// TIA Portal project "SortingStation" (V17)

(* hardware
DEVICE "S7-1500/ET200MP station_1"  S7-1500 station
   slot 0: "Rail_0"  Rack  6ES7 590-1***0-0AA0
   slot 1: "PLC_1"  CPU 1511-1 PN  6ES7 511-1AK02-0AB0  V2.9
      slot 3: "CPU display_1"  6ES7591-1AA00-0AA0
      slot 32768: "PROFINET interface_1"  X1
         slot 32769: "Port_1"  X1 P1
         slot 32770: "Port_2"  X1 P2
      slot 34817: "Virtual CP interface port_1"  Virtual CP interface port  Virtual CP interface port
   slot 2: "DI 16x24VDC BA_1"  DI 16x24VDC BA  6ES7 521-1BH10-0AA0  V1.1
   slot 3: "DQ 16x24VDC/0.5A BA_1"  DQ 16x24VDC/0.5A BA  6ES7 522-1BH10-0AA0  V1.1
   slot 4: "AI 4xU/I/RTD/TC ST_1"  AI 4xU/I/RTD/TC ST  6ES7 531-7QD00-0AB0  V1.0
   slot 5: "AQ 4xU/I ST_1"  AQ 4xU/I ST  6ES7 532-5HD00-0AB0  V2.2
*)

// ===== PLC "PLC_1"  CPU 1511-1 PN =====

VAR_GLOBAL   // PLC tag table "Default tag table"
   "System_Byte" AT %MB1 : Byte;
   "FirstScan" AT %M1.0 : Bool;
   "DiagStatusUpdate" AT %M1.1 : Bool;
   "AlwaysTRUE" AT %M1.2 : Bool;
   "AlwaysFALSE" AT %M1.3 : Bool;
   "Clock_Byte" AT %MB0 : Byte;
   "Clock_10Hz" AT %M0.0 : Bool;
   "Clock_5Hz" AT %M0.1 : Bool;
   "Clock_2.5Hz" AT %M0.2 : Bool;
   "Clock_2Hz" AT %M0.3 : Bool;
   "Clock_1.25Hz" AT %M0.4 : Bool;
   "Clock_1Hz" AT %M0.5 : Bool;
   "Clock_0.625Hz" AT %M0.6 : Bool;
   "Clock_0.5Hz" AT %M0.7 : Bool;
END_VAR

VAR_GLOBAL   // PLC tag table "io"
   "At exit" AT %I0.0 : Bool;
   "Counter 1" AT %QD30 : DInt;
   "Vision sensor" AT %ID30 : DInt;
   "Remover 3" AT %Q1.7 : Bool;
   "Remover 2" AT %Q1.6 : Bool;
   "Remover 1" AT %Q1.5 : Bool;
   "Emitter" AT %Q1.4 : Bool;
   "Stop light" AT %Q1.3 : Bool;
   "Reset light" AT %Q1.2 : Bool;
   "Start light" AT %Q1.1 : Bool;
   "Sorter 3 belt" AT %Q1.0 : Bool;
   "Sorter 3 turn" AT %Q0.7 : Bool;
   "Sorter 2 belt" AT %Q0.6 : Bool;
   "Sorter 2 turn" AT %Q0.5 : Bool;
   "Sorter 1 belt" AT %Q0.4 : Bool;
   "Sorter 1 turn" AT %Q0.3 : Bool;
   "Exit conveyor" AT %Q0.2 : Bool;
   "Stop blade" AT %Q0.1 : Bool;
   "Entry conveyor" AT %Q0.0 : Bool;
   "Manual" AT %I0.7 : Bool;
   "FACTORY I/O (Running)" AT %I0.6 : Bool;
   "Auto" AT %I0.5 : Bool;
   "Emergency stop" AT %I0.4 : Bool;
   "Stop" AT %I0.3 : Bool;
   "Reset" AT %I0.2 : Bool;
   "Start" AT %I0.1 : Bool;
   "Counter 2" AT %QD34 : DInt;
   "Counter 3" AT %QD38 : DInt;
END_VAR

DATA_BLOCK "HmiData"   // DB1
{ S7_Optimized_Access := 'TRUE' }
VERSION : 0.1
   VAR
      Flank : Bool;
      Flank_1 : Bool;
      Flank_2 : Bool;
      Flank_3 : Bool;
      Flank_4 : Bool;
      reset1 : Bool;
      reset2 : Bool;
      reset3 : Bool;
   END_VAR
BEGIN
END_DATA_BLOCK

// folder: System blocks/Program resources

DATA_BLOCK "IEC_Counter_0_DB_3"   // DB5
{ S7_Optimized_Access := 'TRUE' }
AUTHOR : Simatic
FAMILY : IEC
NAME : CNTR
VERSION : 1.0
// stored: InstanceOfName IEC_COUNTER
"IEC_COUNTER"
BEGIN
END_DATA_BLOCK

DATA_BLOCK "IEC_Counter_0_DB_4"   // DB6
{ S7_Optimized_Access := 'TRUE' }
AUTHOR : Simatic
FAMILY : IEC
NAME : CNTR
VERSION : 1.0
// stored: InstanceOfName IEC_COUNTER
"IEC_COUNTER"
BEGIN
END_DATA_BLOCK

DATA_BLOCK "IEC_Counter_0_DB_5"   // DB7
{ S7_Optimized_Access := 'TRUE' }
AUTHOR : Simatic
FAMILY : IEC
NAME : CNTR
VERSION : 1.0
// stored: InstanceOfName IEC_COUNTER
"IEC_COUNTER"
BEGIN
END_DATA_BLOCK

// folder: (top level)

FUNCTION "Hmi" : Void   // FC1, LAD
{ S7_Optimized_Access := 'TRUE' }
VERSION : 0.1
   VAR_TEMP   // added for the SCL form of the ladder/FBD networks
      _w1 : Bool;
   END_VAR
BEGIN

REGION Network 1: Start logik
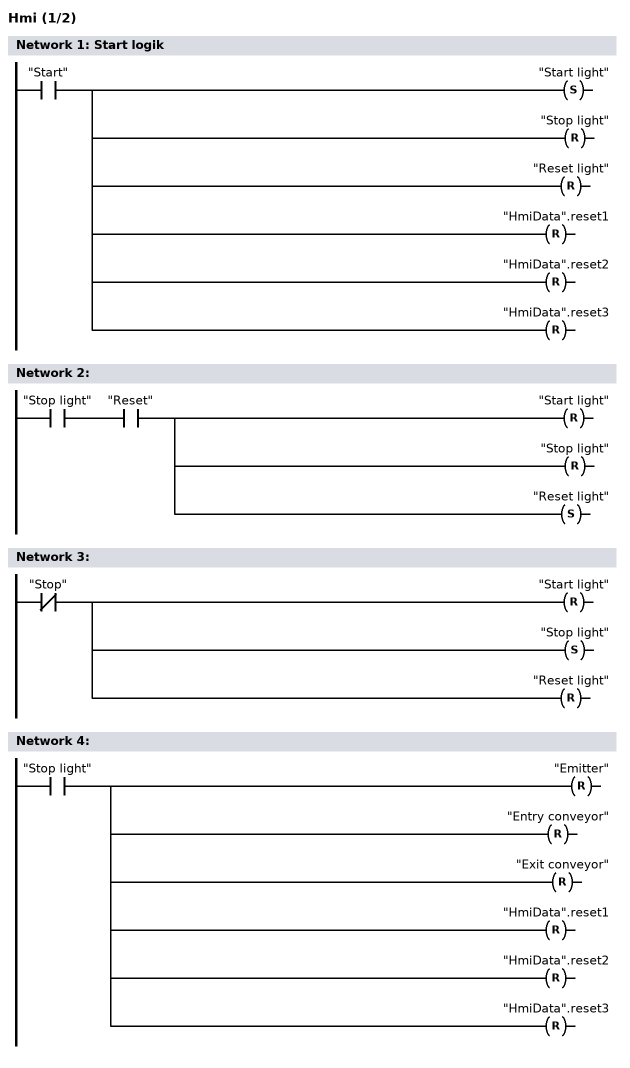
   RUNG wire#powerrail
      Contact( "Start" )
      wire#w1
      S_Coil( "Start light" )
   END_RUNG
   RUNG wire#w1
      R_Coil( "Stop light" )
   END_RUNG
   RUNG wire#w1
      R_Coil( "Reset light" )
   END_RUNG
   RUNG wire#w1
      R_Coil( "HmiData".reset1 )
   END_RUNG
   RUNG wire#w1
      R_Coil( "HmiData".reset2 )
   END_RUNG
   RUNG wire#w1
      R_Coil( "HmiData".reset3 )
   END_RUNG
   // the same network as SCL:
   IF "Start" THEN
       "Start light" := TRUE;
       "Stop light" := FALSE;
       "Reset light" := FALSE;
       "HmiData".reset1 := FALSE;
       "HmiData".reset2 := FALSE;
       "HmiData".reset3 := FALSE;
   END_IF;
END_REGION

REGION Network 2
   RUNG wire#powerrail
      Contact( "Stop light" )
      Contact( "Reset" )
      wire#w1
      R_Coil( "Start light" )
   END_RUNG
   RUNG wire#w1
      R_Coil( "Stop light" )
   END_RUNG
   RUNG wire#w1
      S_Coil( "Reset light" )
   END_RUNG
   // the same network as SCL:
   IF "Stop light" AND "Reset" THEN "Start light" := FALSE; END_IF;
   #_w1 := "Stop light" AND "Reset";
   IF #_w1 THEN
       "Stop light" := FALSE;
       "Reset light" := TRUE;
   END_IF;
END_REGION

REGION Network 3
   RUNG wire#powerrail
      I_Contact( "Stop" )
      wire#w1
      R_Coil( "Start light" )
   END_RUNG
   RUNG wire#w1
      S_Coil( "Stop light" )
   END_RUNG
   RUNG wire#w1
      R_Coil( "Reset light" )
   END_RUNG
   // the same network as SCL:
   IF NOT "Stop" THEN
       "Start light" := FALSE;
       "Stop light" := TRUE;
       "Reset light" := FALSE;
   END_IF;
END_REGION

REGION Network 4
   RUNG wire#powerrail
      Contact( "Stop light" )
      wire#w1
      R_Coil( "Emitter" )
   END_RUNG
   RUNG wire#w1
      R_Coil( "Entry conveyor" )
   END_RUNG
   RUNG wire#w1
      R_Coil( "Exit conveyor" )
   END_RUNG
   RUNG wire#w1
      R_Coil( "HmiData".reset1 )
   END_RUNG
   RUNG wire#w1
      R_Coil( "HmiData".reset2 )
   END_RUNG
   RUNG wire#w1
      R_Coil( "HmiData".reset3 )
   END_RUNG
   // the same network as SCL:
   IF "Stop light" THEN
       "Emitter" := FALSE;
       "Entry conveyor" := FALSE;
       "Exit conveyor" := FALSE;
       "HmiData".reset1 := FALSE;
       "HmiData".reset2 := FALSE;
       "HmiData".reset3 := FALSE;
   END_IF;
END_REGION

REGION Network 5
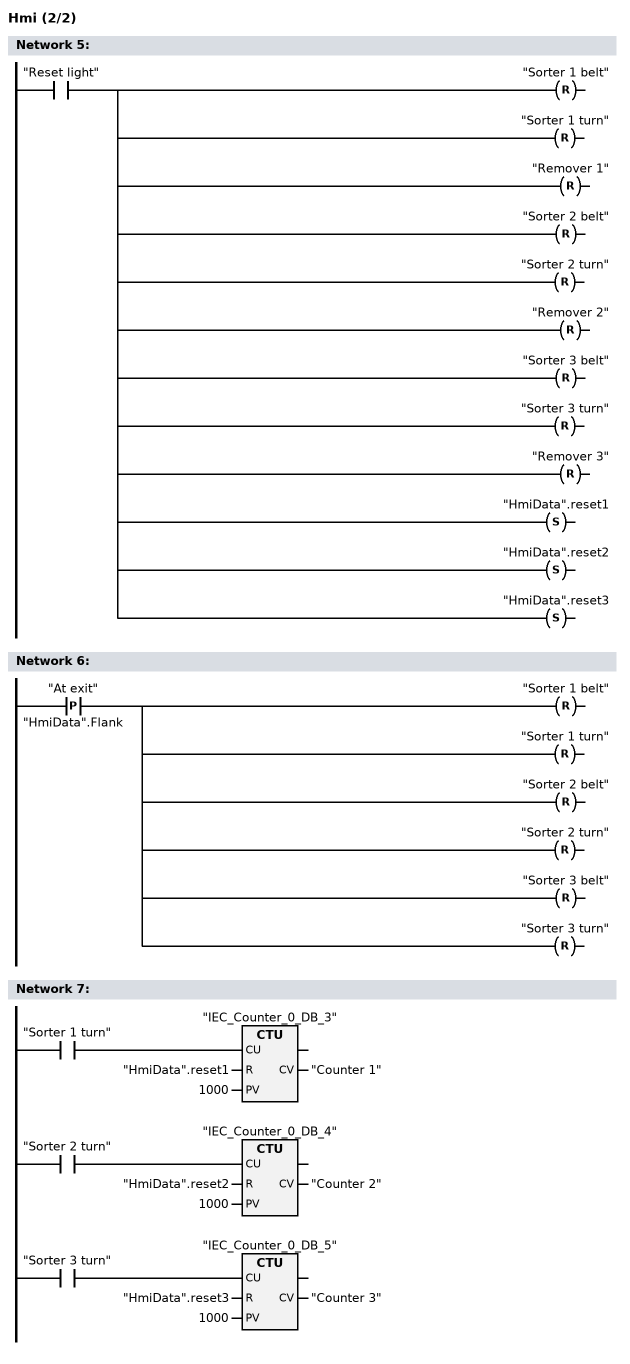
   RUNG wire#powerrail
      Contact( "Reset light" )
      wire#w1
      R_Coil( "Sorter 1 belt" )
   END_RUNG
   RUNG wire#w1
      R_Coil( "Sorter 1 turn" )
   END_RUNG
   RUNG wire#w1
      R_Coil( "Remover 1" )
   END_RUNG
   RUNG wire#w1
      R_Coil( "Sorter 2 belt" )
   END_RUNG
   RUNG wire#w1
      R_Coil( "Sorter 2 turn" )
   END_RUNG
   RUNG wire#w1
      R_Coil( "Remover 2" )
   END_RUNG
   RUNG wire#w1
      R_Coil( "Sorter 3 belt" )
   END_RUNG
   RUNG wire#w1
      R_Coil( "Sorter 3 turn" )
   END_RUNG
   RUNG wire#w1
      R_Coil( "Remover 3" )
   END_RUNG
   RUNG wire#w1
      S_Coil( "HmiData".reset1 )
   END_RUNG
   RUNG wire#w1
      S_Coil( "HmiData".reset2 )
   END_RUNG
   RUNG wire#w1
      S_Coil( "HmiData".reset3 )
   END_RUNG
   // the same network as SCL:
   IF "Reset light" THEN
       "Sorter 1 belt" := FALSE;
       "Sorter 1 turn" := FALSE;
       "Remover 1" := FALSE;
       "Sorter 2 belt" := FALSE;
       "Sorter 2 turn" := FALSE;
       "Remover 2" := FALSE;
       "Sorter 3 belt" := FALSE;
       "Sorter 3 turn" := FALSE;
       "Remover 3" := FALSE;
       "HmiData".reset1 := TRUE;
       "HmiData".reset2 := TRUE;
       "HmiData".reset3 := TRUE;
   END_IF;
END_REGION

REGION Network 6
   RUNG wire#powerrail
      P_Contact(operand := "At exit", bit := "HmiData".Flank)
      wire#w1
      R_Coil( "Sorter 1 belt" )
   END_RUNG
   RUNG wire#w1
      R_Coil( "Sorter 1 turn" )
   END_RUNG
   RUNG wire#w1
      R_Coil( "Sorter 2 belt" )
   END_RUNG
   RUNG wire#w1
      R_Coil( "Sorter 2 turn" )
   END_RUNG
   RUNG wire#w1
      R_Coil( "Sorter 3 belt" )
   END_RUNG
   RUNG wire#w1
      R_Coil( "Sorter 3 turn" )
   END_RUNG
   // the same network as SCL:
   #_w1 := "At exit" AND NOT "HmiData".Flank;   // rising edge of "At exit"
   "HmiData".Flank := "At exit";
   IF #_w1 THEN
       "Sorter 1 belt" := FALSE;
       "Sorter 1 turn" := FALSE;
       "Sorter 2 belt" := FALSE;
       "Sorter 2 turn" := FALSE;
       "Sorter 3 belt" := FALSE;
       "Sorter 3 turn" := FALSE;
   END_IF;
END_REGION

REGION Network 7
   "IEC_Counter_0_DB_3".CTU(CU := "Sorter 1 turn", R := "HmiData".reset1, PV := 1000, CV => "Counter 1");
   "IEC_Counter_0_DB_4".CTU(CU := "Sorter 2 turn", R := "HmiData".reset2, PV := 1000, CV => "Counter 2");
   "IEC_Counter_0_DB_5".CTU(CU := "Sorter 3 turn", R := "HmiData".reset3, PV := 1000, CV => "Counter 3");
END_REGION
END_FUNCTION

FUNCTION "Kör programmet" : Void   // FC2, LAD
{ S7_Optimized_Access := 'TRUE' }
VERSION : 0.1
BEGIN

REGION Network 1
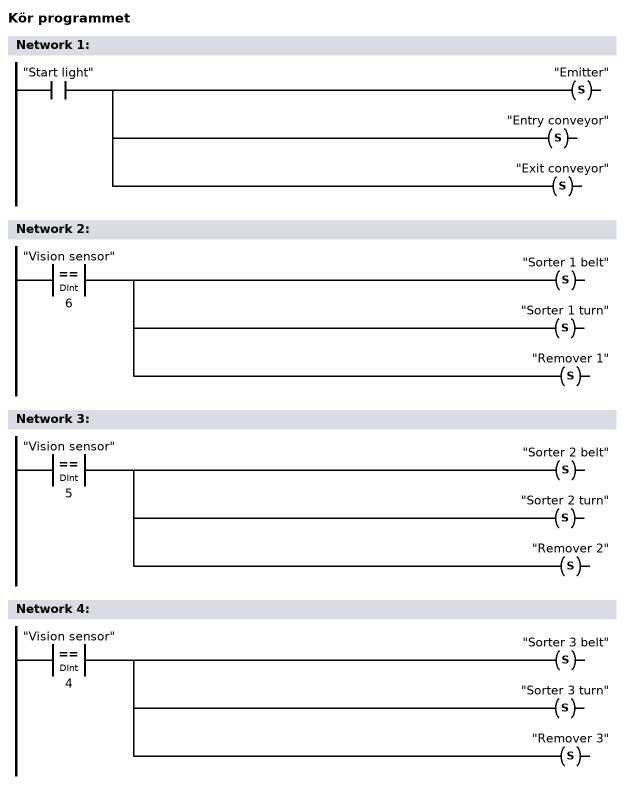
   RUNG wire#powerrail
      Contact( "Start light" )
      wire#w1
      S_Coil( "Emitter" )
   END_RUNG
   RUNG wire#w1
      S_Coil( "Entry conveyor" )
   END_RUNG
   RUNG wire#w1
      S_Coil( "Exit conveyor" )
   END_RUNG
   // the same network as SCL:
   IF "Start light" THEN
       "Emitter" := TRUE;
       "Entry conveyor" := TRUE;
       "Exit conveyor" := TRUE;
   END_IF;
END_REGION

REGION Network 2
   RUNG wire#powerrail
      { S7_Templates := "SrcType := DInt" } EQ_Contact(in1 := "Vision sensor", in2 := 6)
      wire#w1
      S_Coil( "Sorter 1 belt" )
   END_RUNG
   RUNG wire#w1
      S_Coil( "Sorter 1 turn" )
   END_RUNG
   RUNG wire#w1
      S_Coil( "Remover 1" )
   END_RUNG
   // the same network as SCL:
   IF "Vision sensor" = 6 THEN
       "Sorter 1 belt" := TRUE;
       "Sorter 1 turn" := TRUE;
       "Remover 1" := TRUE;
   END_IF;
END_REGION

REGION Network 3
   RUNG wire#powerrail
      { S7_Templates := "SrcType := DInt" } EQ_Contact(in1 := "Vision sensor", in2 := 5)
      wire#w1
      S_Coil( "Sorter 2 belt" )
   END_RUNG
   RUNG wire#w1
      S_Coil( "Sorter 2 turn" )
   END_RUNG
   RUNG wire#w1
      S_Coil( "Remover 2" )
   END_RUNG
   // the same network as SCL:
   IF "Vision sensor" = 5 THEN
       "Sorter 2 belt" := TRUE;
       "Sorter 2 turn" := TRUE;
       "Remover 2" := TRUE;
   END_IF;
END_REGION

REGION Network 4
   RUNG wire#powerrail
      { S7_Templates := "SrcType := DInt" } EQ_Contact(in1 := "Vision sensor", in2 := 4)
      wire#w1
      S_Coil( "Sorter 3 belt" )
   END_RUNG
   RUNG wire#w1
      S_Coil( "Sorter 3 turn" )
   END_RUNG
   RUNG wire#w1
      S_Coil( "Remover 3" )
   END_RUNG
   // the same network as SCL:
   IF "Vision sensor" = 4 THEN
       "Sorter 3 belt" := TRUE;
       "Sorter 3 turn" := TRUE;
       "Remover 3" := TRUE;
   END_IF;
END_REGION
END_FUNCTION

ORGANIZATION_BLOCK "Main"   // OB1, LAD, ProgramCycle
TITLE = "Main Program Sweep (Cycle)"
{ S7_Optimized_Access := 'TRUE' }
VERSION : 0.1
   VAR_INPUT
      Initial_Call : Bool;   // Initial call of this OB
      Remanence : Bool;   // =True, if remanent data are available
   END_VAR
BEGIN

REGION Network 1
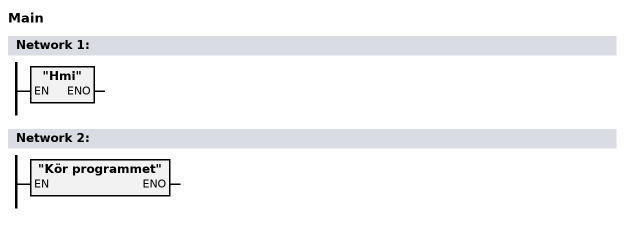
   RUNG wire#powerrail
      "Hmi"()
   END_RUNG
   // the same network as SCL:
   "Hmi"();
END_REGION

REGION Network 2
   RUNG wire#powerrail
      "Kör programmet"()
   END_RUNG
   // the same network as SCL:
   "Kör programmet"();
END_REGION
END_ORGANIZATION_BLOCK